DATA_BLOCK "tcp"
{ S7_Optimized_Access := 'FALSE' }
VERSION : 0.1
NON_RETAIN
"modbus_tcp_new"

BEGIN

END_DATA_BLOCK

